FUNCTION_BLOCK FB_FT_IMP (* Composite Function Block Type *)
  (* Standard: 61499-2 *)
  (* Version 0.0, 2011-08-27, 4DIAC-IDE, 4DIAC-Consortium *)
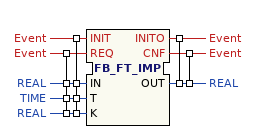
  EVENT_INPUT
    INIT WITH T, K, IN; (* Initialization Request *)
    REQ WITH IN, T, K; (* Normal Execution Request *)
  END_EVENT
  EVENT_OUTPUT
    INITO WITH OUT; (* Initialization Confirm *)
    CNF WITH OUT; (* Execution Confirmation *)
  END_EVENT
  VAR_INPUT
    IN : REAL; (* input signal *)
    T : TIME; (* time constant *)
    K : REAL := 1.0; (* multiplier *)
  END_VAR
  VAR_OUTPUT
    OUT : REAL; (* high pass with time constant T *)
  END_VAR
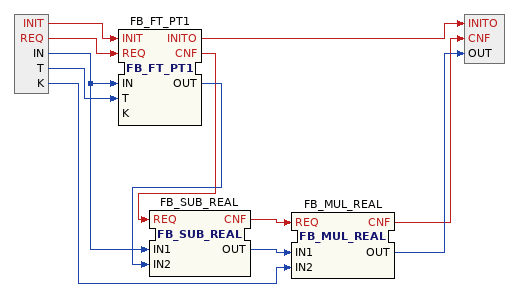
  FBS
    FB_FT_PT1 : FB_FT_PT1;
    FB_MUL_REAL : FB_MUL_REAL;
    FB_SUB_REAL : FB_SUB_REAL;
  END_FBS
  EVENT_CONNECTIONS
    INIT TO FB_FT_PT1.INIT;
    FB_FT_PT1.INITO TO INITO;
    REQ TO FB_FT_PT1.REQ;
    FB_FT_PT1.CNF TO FB_SUB_REAL.REQ;
    FB_SUB_REAL.CNF TO FB_MUL_REAL.REQ;
    FB_MUL_REAL.CNF TO CNF;
  END_CONNECTIONS
  DATA_CONNECTIONS
    IN TO FB_FT_PT1.IN;
    T TO FB_FT_PT1.T;
    IN TO FB_SUB_REAL.IN1;
    FB_FT_PT1.OUT TO FB_SUB_REAL.IN2;
    FB_SUB_REAL.OUT TO FB_MUL_REAL.IN1;
    K TO FB_MUL_REAL.IN2;
    FB_MUL_REAL.OUT TO OUT;
  END_CONNECTIONS
END_FUNCTION_BLOCK
